(* PLC project RedHat_Demo_MarketingStand_Working.project, CODESYS CODESYS V3.5 SP22 *)
(* stored: creationDateTime 2026-08-06T19:18:19.3184089, modificationDateTime 2026-08-06T19:18:02.9898727 *)

PROGRAM PLC_PRG
  VAR
    Cmd_Run : BOOL;
    R_TRIG_0 : R_TRIG;
    Sequence_Run : DINT := 0;
    Sts_SequenceDone : BOOL;
    Sts_FirstScanBit : BOOL := TRUE;
    TON_MotorDataDelay : ARRAY[0..9] OF TON;
    TON_IndexPauseDelay : TON;
    Par_IndexPause : TIME := TIME#1s0ms;
    TON_Timeout_Reset : TON;
    TON_Timeout_Enable : TON;
    TON_Timeout_Move1 : TON;
    TON_Timeout_Move2 : TON;
    TON_Timeout_Stop : TON;
    Sts_SeqTimeout : DINT;
    Force_Run : BOOL;
    Force_Stop : BOOL;
    Cmd_Stop : BOOL;
    Par_SingleIndex : BOOL;
    TimeStart1 : LTIME;
    tDelta : TIME;
    tStart : TIME;
    tEnd : TIME;
    Return_Time_Input : BOOL;
    ReturnTimeFinish : BOOL;
    MoveDelta : BOOL;
    newTimeDelta : TIME;
    IndexPauseInt : REAL;
    IndexPauseMin : REAL := 500;
    IndexPauseMax : REAL := 5000;
    RealTimeDelta : REAL;
    microtime : SYSTIME;
    Seq0 : BOOL;
    Seq10 : BOOL;
    Seq20 : BOOL;
    Seq30 : BOOL;
    Seq40 : BOOL;
    Seq50 : BOOL;
    Seq60 : BOOL;
    SeqErr : BOOL;
    MotorEnabled : BOOL;
    SeqStop : BOOL;
    SeqMov1 : BOOL;
    SeqMov2 : BOOL;
  END_VAR
  VAR  (* added by the conversion: wires and edge detectors of the diagram *)
    _NE7_OUT : BOOL;
    _EQ14_ENO : BOOL;
    _EQ14_OUT : BOOL;
    _w20 : BOOL;
    _w21 : BOOL;
    _EQ27_ENO : BOOL;
    _EQ27_OUT : BOOL;
    _EQ35_OUT : BOOL;
    _EQ48_OUT : BOOL;
    _EQ65_OUT : BOOL;
    _EQ76_OUT : BOOL;
    _EQ93_OUT : BOOL;
    _EQ113_OUT : BOOL;
    _EQ130_OUT : BOOL;
    _MOVE138_EN : BOOL;
    _EQ145_OUT : BOOL;
    _MOVE162_EN : BOOL;
    R_TRIG1 : R_TRIG;
    R_TRIG2 : R_TRIG;
    _FUNC_SCALE196_EN : BOOL;
  END_VAR

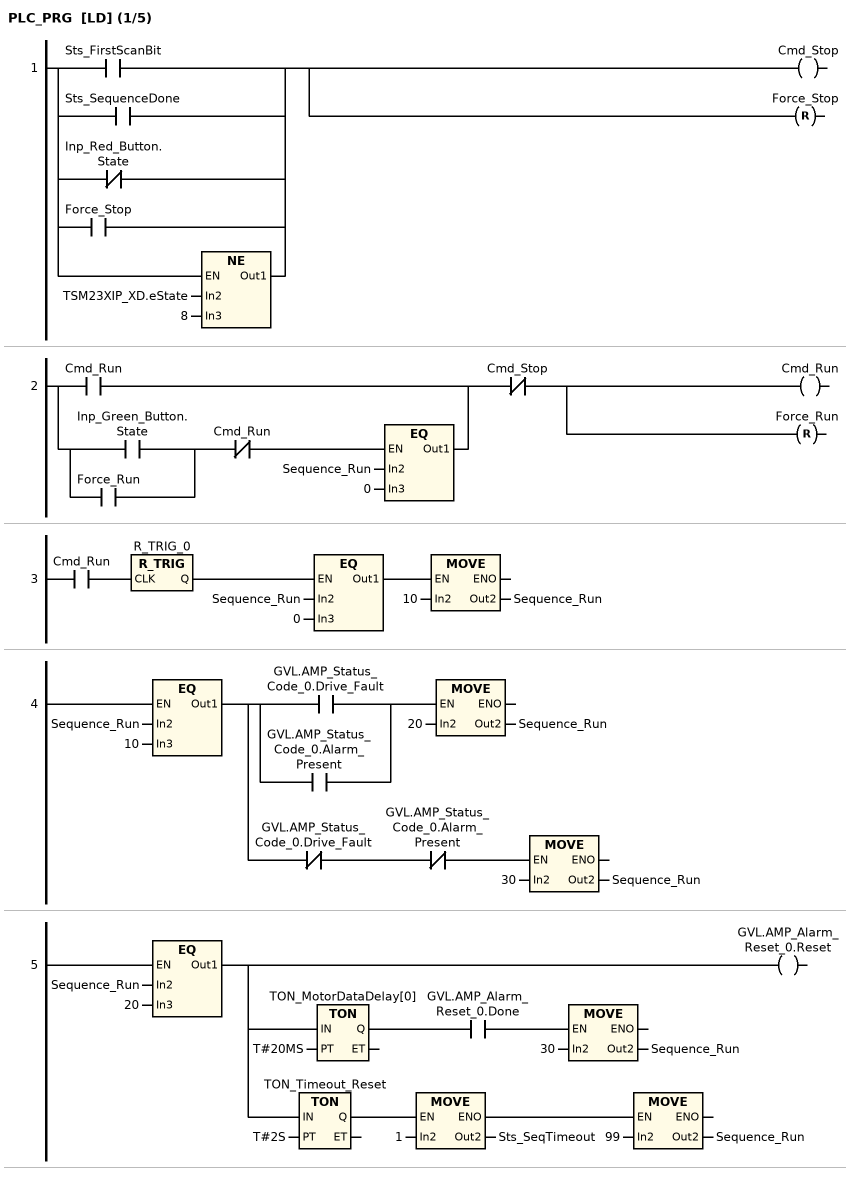
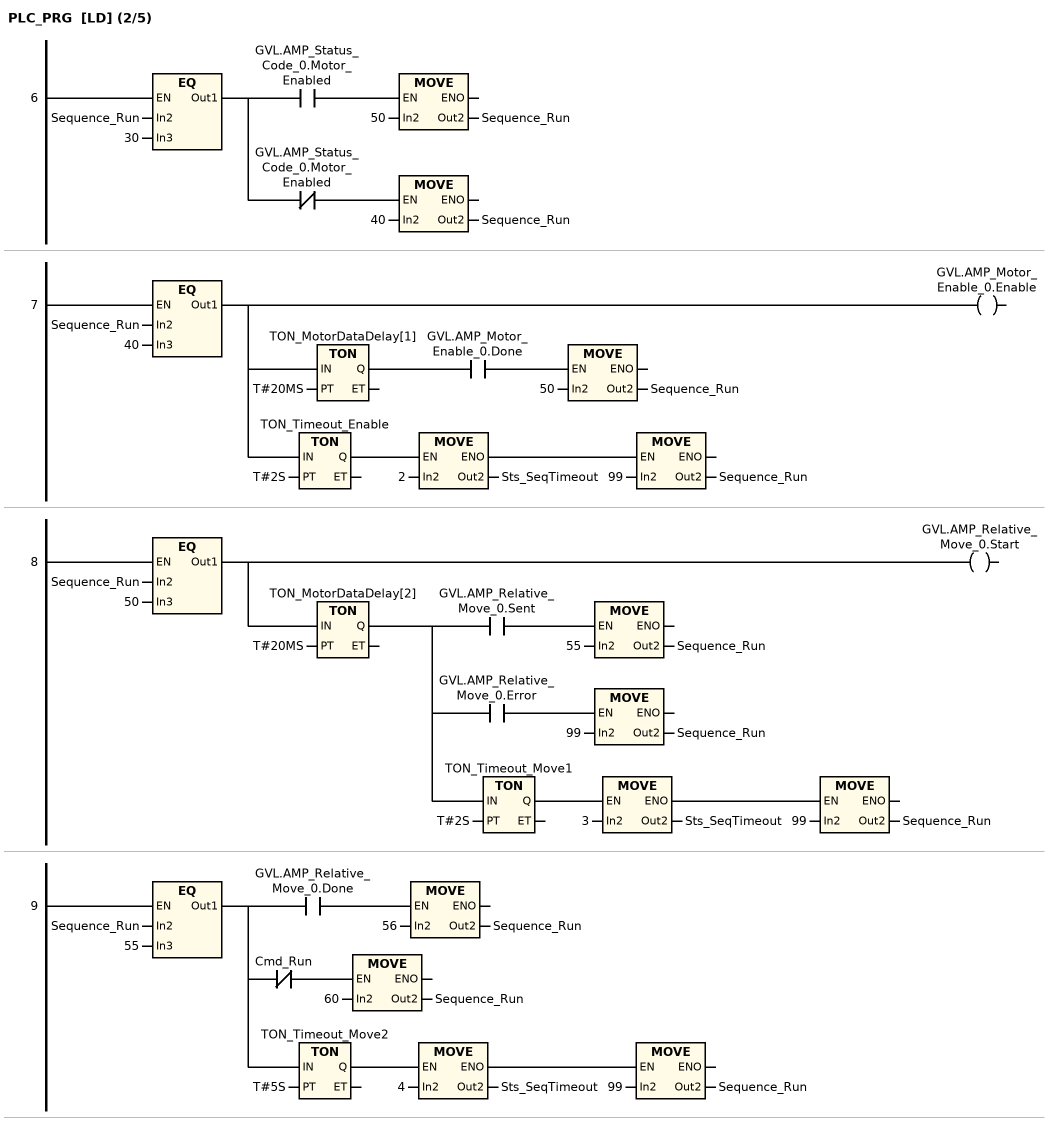
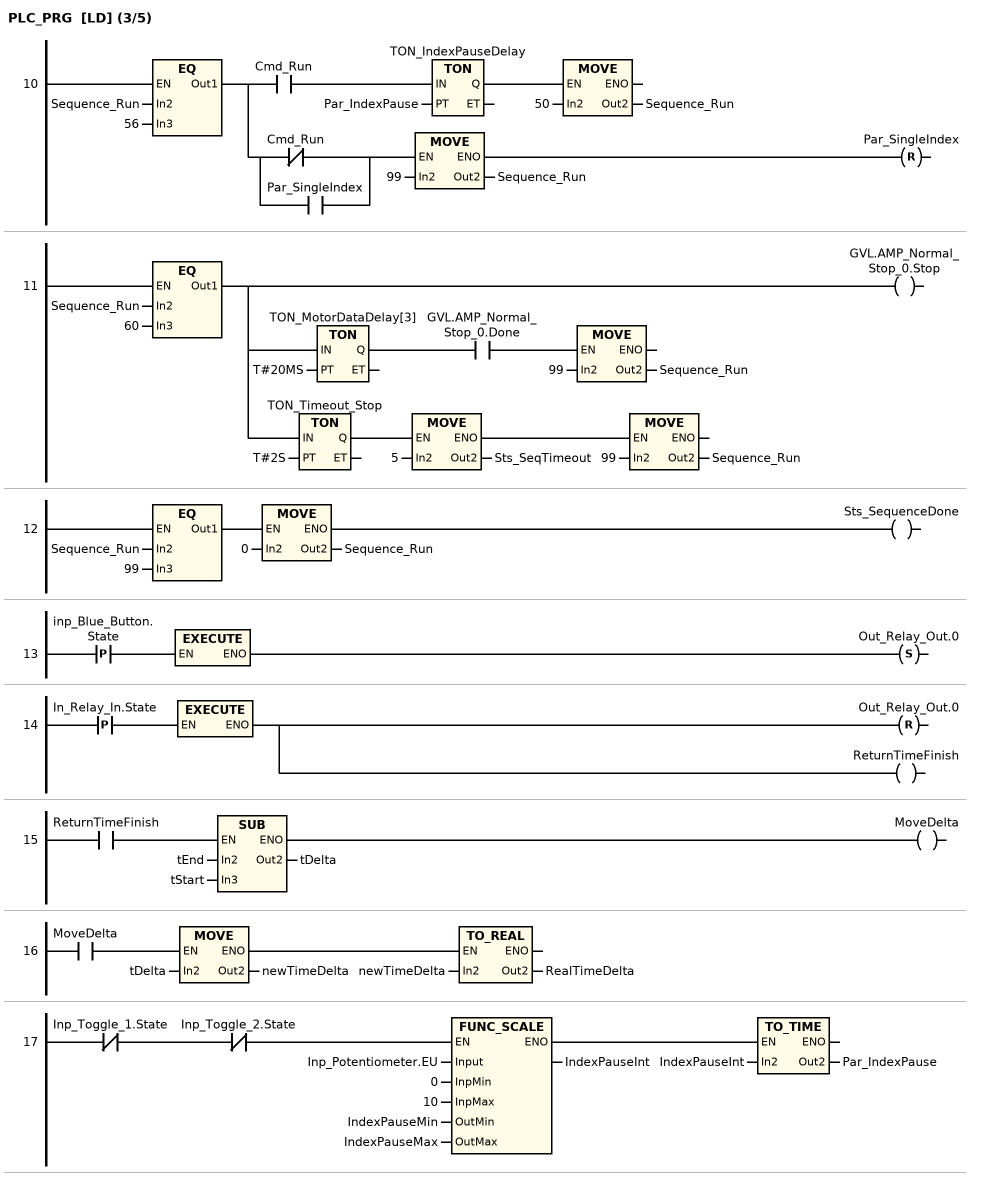
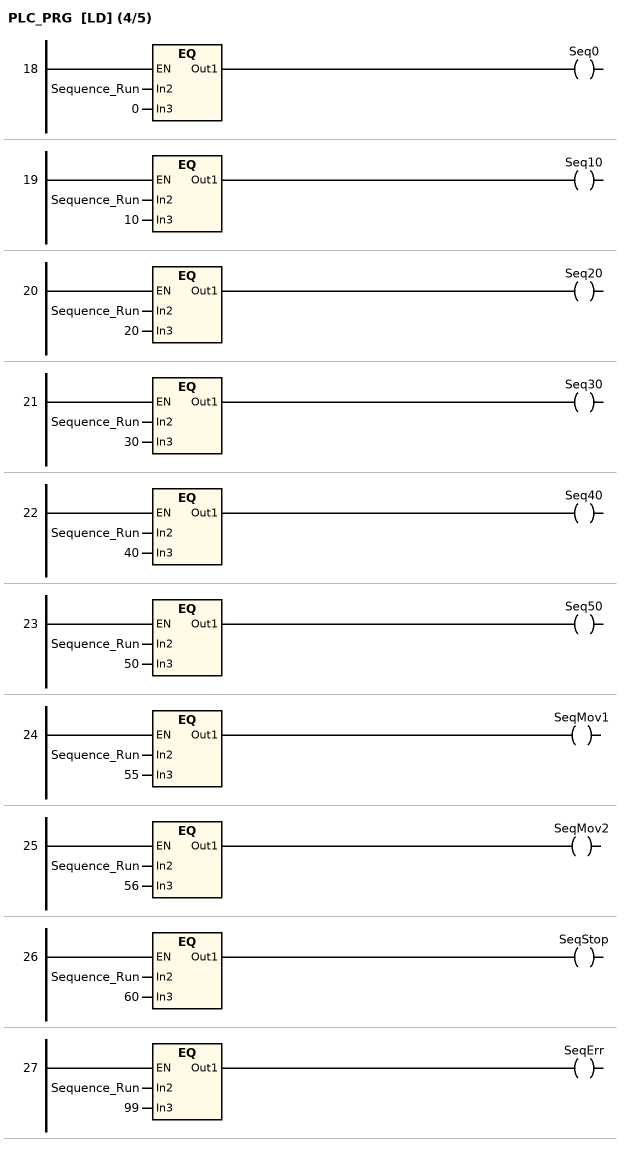
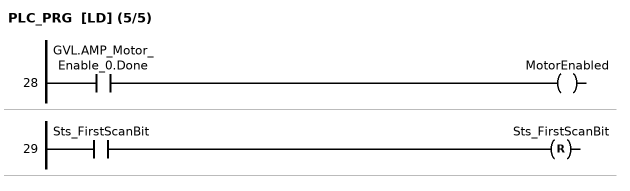
(* LD diagram, written out as Structured Text *)
(* Run Permissives *)

_NE7_OUT := TSM23XIP_XD.eState <> 8;
Cmd_Stop := Sts_FirstScanBit OR Sts_SequenceDone OR NOT Inp_Red_Button.State OR Force_Stop OR _NE7_OUT;
IF Sts_FirstScanBit OR Sts_SequenceDone OR NOT Inp_Red_Button.State OR Force_Stop OR _NE7_OUT THEN Force_Stop := FALSE; END_IF;
(* Start Sequence Command *)

_EQ14_OUT := EQ(EN := (Inp_Green_Button.State OR Force_Run) AND NOT Cmd_Run, IN1 := Sequence_Run, IN2 := 0, ENO => _EQ14_ENO);
_w20 := Cmd_Run;
_w21 := (_EQ14_OUT OR _w20) AND NOT Cmd_Stop;
Cmd_Run := _w21;
IF _w21 THEN Force_Run := FALSE; END_IF;

R_TRIG_0(CLK := Cmd_Run);
_EQ27_OUT := EQ(EN := R_TRIG_0.Q, IN1 := Sequence_Run, IN2 := 0, ENO => _EQ27_ENO);
IF _EQ27_OUT THEN Sequence_Run := 10; END_IF;

_EQ35_OUT := Sequence_Run = 10;
IF _EQ35_OUT AND NOT GVL.AMP_Status_Code_0.Drive_Fault AND NOT GVL.AMP_Status_Code_0.Alarm_Present THEN Sequence_Run := 30; END_IF;
IF _EQ35_OUT AND (GVL.AMP_Status_Code_0.Drive_Fault OR GVL.AMP_Status_Code_0.Alarm_Present) THEN Sequence_Run := 20; END_IF;
(* Fault Reset *)

_EQ48_OUT := Sequence_Run = 20;
GVL.AMP_Alarm_Reset_0.Reset := _EQ48_OUT;
TON_MotorDataDelay[0](IN := _EQ48_OUT, PT := T#20MS);
IF TON_MotorDataDelay[0].Q AND GVL.AMP_Alarm_Reset_0.Done THEN Sequence_Run := 30; END_IF;
TON_Timeout_Reset(IN := _EQ48_OUT, PT := T#2S);
IF TON_Timeout_Reset.Q THEN Sts_SeqTimeout := 1; END_IF;
IF TON_Timeout_Reset.Q THEN Sequence_Run := 99; END_IF;

_EQ65_OUT := Sequence_Run = 30;
IF _EQ65_OUT AND GVL.AMP_Status_Code_0.Motor_Enabled THEN Sequence_Run := 50; END_IF;
IF _EQ65_OUT AND NOT GVL.AMP_Status_Code_0.Motor_Enabled THEN Sequence_Run := 40; END_IF;
(* Energize *)

_EQ76_OUT := Sequence_Run = 40;
GVL.AMP_Motor_Enable_0.Enable := _EQ76_OUT;
TON_MotorDataDelay[1](IN := _EQ76_OUT, PT := T#20MS);
IF TON_MotorDataDelay[1].Q AND GVL.AMP_Motor_Enable_0.Done THEN Sequence_Run := 50; END_IF;
TON_Timeout_Enable(IN := _EQ76_OUT, PT := T#2S);
IF TON_Timeout_Enable.Q THEN Sts_SeqTimeout := 2; END_IF;
IF TON_Timeout_Enable.Q THEN Sequence_Run := 99; END_IF;
(* Incremental Move *)

_EQ93_OUT := Sequence_Run = 50;
GVL.AMP_Relative_Move_0.Start := _EQ93_OUT;
TON_MotorDataDelay[2](IN := _EQ93_OUT, PT := T#20MS);
IF TON_MotorDataDelay[2].Q AND GVL.AMP_Relative_Move_0.Sent THEN Sequence_Run := 55; END_IF;
IF TON_MotorDataDelay[2].Q AND GVL.AMP_Relative_Move_0.Error THEN Sequence_Run := 99; END_IF;
TON_Timeout_Move1(IN := TON_MotorDataDelay[2].Q, PT := T#2S);
IF TON_Timeout_Move1.Q THEN Sts_SeqTimeout := 3; END_IF;
IF TON_Timeout_Move1.Q THEN Sequence_Run := 99; END_IF;
(* Wait For Move To Complete, or Stop button Press *)

_EQ113_OUT := Sequence_Run = 55;
IF _EQ113_OUT AND GVL.AMP_Relative_Move_0.Done THEN Sequence_Run := 56; END_IF;
IF _EQ113_OUT AND NOT Cmd_Run THEN Sequence_Run := 60; END_IF;
TON_Timeout_Move2(IN := _EQ113_OUT, PT := T#5S);
IF TON_Timeout_Move2.Q THEN Sts_SeqTimeout := 4; END_IF;
IF TON_Timeout_Move2.Q THEN Sequence_Run := 99; END_IF;
(* Pause before next index (Loop Up) *)

_EQ130_OUT := Sequence_Run = 56;
TON_IndexPauseDelay(IN := _EQ130_OUT AND Cmd_Run, PT := Par_IndexPause);
IF TON_IndexPauseDelay.Q THEN Sequence_Run := 50; END_IF;
_MOVE138_EN := _EQ130_OUT AND (NOT Cmd_Run OR Par_SingleIndex);
IF _MOVE138_EN THEN Sequence_Run := 99; END_IF;
IF _MOVE138_EN THEN Par_SingleIndex := FALSE; END_IF;
(* Normal Stop *)

_EQ145_OUT := Sequence_Run = 60;
GVL.AMP_Normal_Stop_0.Stop := _EQ145_OUT;
TON_MotorDataDelay[3](IN := _EQ145_OUT, PT := T#20MS);
IF TON_MotorDataDelay[3].Q AND GVL.AMP_Normal_Stop_0.Done THEN Sequence_Run := 99; END_IF;
TON_Timeout_Stop(IN := _EQ145_OUT, PT := T#2S);
IF TON_Timeout_Stop.Q THEN Sts_SeqTimeout := 5; END_IF;
IF TON_Timeout_Stop.Q THEN Sequence_Run := 99; END_IF;
(* Sequence Complete *)

_MOVE162_EN := Sequence_Run = 99;
IF _MOVE162_EN THEN Sequence_Run := 0; END_IF;
Sts_SequenceDone := _MOVE162_EN;

R_TRIG1(CLK := inp_Blue_Button.State);
IF R_TRIG1.Q THEN
  tStart := TO_TIME(SysTimeGetMs());
END_IF;
IF R_TRIG1.Q THEN Out_Relay_Out.0 := TRUE; END_IF;

R_TRIG2(CLK := In_Relay_In.State);
IF R_TRIG2.Q THEN
  tEnd := TO_TIME(SysTimeGetMs());
END_IF;
IF R_TRIG2.Q THEN Out_Relay_Out.0 := FALSE; END_IF;
ReturnTimeFinish := R_TRIG2.Q;

IF ReturnTimeFinish THEN tDelta := tEnd - tStart; END_IF;
MoveDelta := ReturnTimeFinish;

IF MoveDelta THEN newTimeDelta := tDelta; END_IF;
IF MoveDelta THEN RealTimeDelta := TO_REAL(In2 := newTimeDelta); END_IF;

_FUNC_SCALE196_EN := NOT Inp_Toggle_1.State AND NOT Inp_Toggle_2.State;
IF _FUNC_SCALE196_EN THEN IndexPauseInt := FUNC_SCALE(Input := Inp_Potentiometer.EU, InpMin := 0, InpMax := 10, OutMin := IndexPauseMin, OutMax := IndexPauseMax); END_IF;
IF _FUNC_SCALE196_EN THEN Par_IndexPause := TO_TIME(In2 := IndexPauseInt); END_IF;

Seq0 := Sequence_Run = 0;

Seq10 := Sequence_Run = 10;

Seq20 := Sequence_Run = 20;

Seq30 := Sequence_Run = 30;

Seq40 := Sequence_Run = 40;

Seq50 := Sequence_Run = 50;

SeqMov1 := Sequence_Run = 55;

SeqMov2 := Sequence_Run = 56;


SeqStop := Sequence_Run = 60;

SeqErr := Sequence_Run = 99;

MotorEnabled := GVL.AMP_Motor_Enable_0.Done;

(* Turn off First Scan Bit *)

IF Sts_FirstScanBit THEN Sts_FirstScanBit := FALSE; END_IF;
END_PROGRAM

FUNCTION FUNC_SCALE : REAL
  VAR_INPUT
    Input : REAL;
    InpMin : REAL;
    InpMax : REAL;
    OutMin : REAL;
    OutMax : REAL;
  END_VAR
  VAR
    Value : REAL;
  END_VAR

                    IF Input < InpMin THEN
	Value:= InpMin;
ELSIF Input > InpMax THEN
	Value:= InpMax;
ELSE
	Value:= Input;
END_IF
FUNC_SCALE:= (Value-InpMin) * (OutMax-OutMin) / (InpMax-InpMin) + OutMin;
                  
END_FUNCTION

PROGRAM MOTOR
  VAR CONSTANT
    StepsPerRotation : REAL := 20000;
  END_VAR
  VAR
    Par_SelectorDistance1_Degrees : REAL := -30;  (* Motor Distance variables corresponding to the 3 positions of the selector switch, in degrees. Code converts to steps *)
    Par_SelectorDistance2_Degrees : REAL := 30;
    Par_SelectorDistance3_Degrees : REAL := 60;
    Par_SoftwareDistanceEnable : BOOL;  (* If want to ignore selector switch and use software Distance value *)
    Par_SoftwareDistance_Degrees : REAL;
    MotorDistance_Steps : REAL;  (* Calculated steps to send to motor *)
    Par_PotentiometerMinSpeed : REAL := 0.2;  (* Potentiometer used for index speed. Set minimum and maximum *)
    Par_PotentiometerMaxSpeed : REAL := 0.3;
    Par_AccelDeccel : REAL := 0.167;  (* Constant acceleration and deceleration *)
    Par_SoftwareSpeedEnable : BOOL;  (* If want to ignore potentiometer and use software Speed value *)
    Par_SoftwareSpeed : REAL;
    EncoderPosition_Degrees : REAL;  (* Calculated Position In Degrees of the encoder *)
    Par_SCL_Reg1 : DINT;
    Cmd_ZeroPosition : BOOL;  (* Zero Position Sequence *)
    Sequence_ZeroPosition : DINT;
    TON_MotorDataDelay : ARRAY[0..1] OF TON;
  END_VAR
  VAR  (* added by the conversion: wires and edge detectors of the diagram *)
    _GT46_ENO : BOOL;
    _GT46_OUT : BOOL;
    _EQ103_ENO : BOOL;
    _EQ103_OUT : BOOL;
    _EQ111_OUT : BOOL;
    _EQ121_OUT : BOOL;
    _EQ129_OUT : BOOL;
    _EQ139_OUT : BOOL;
  END_VAR

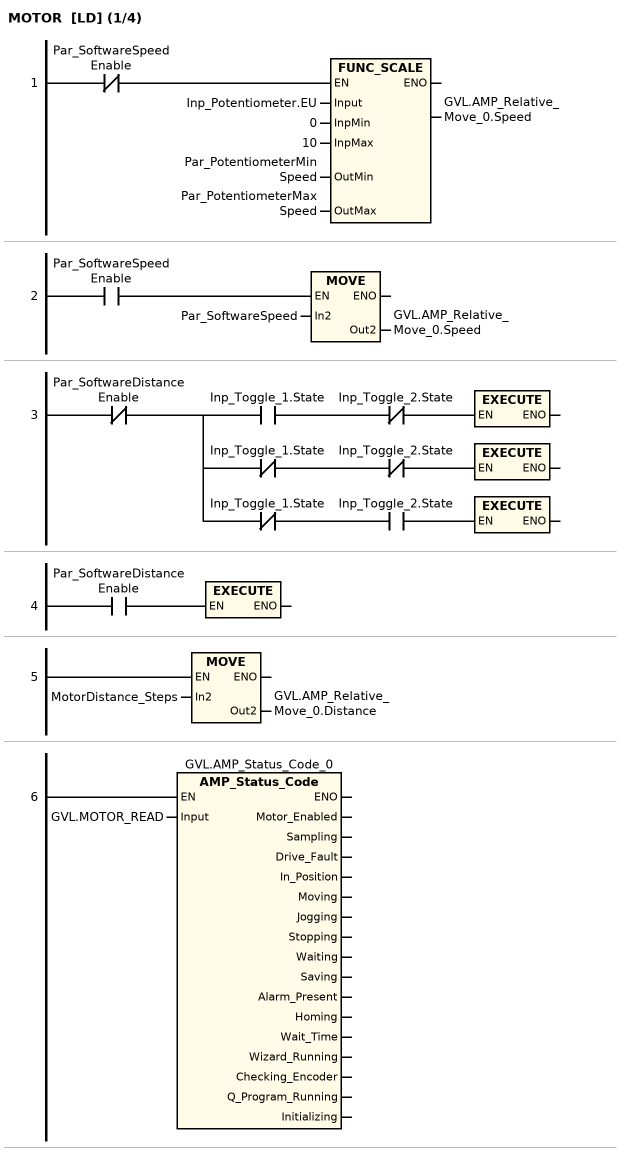
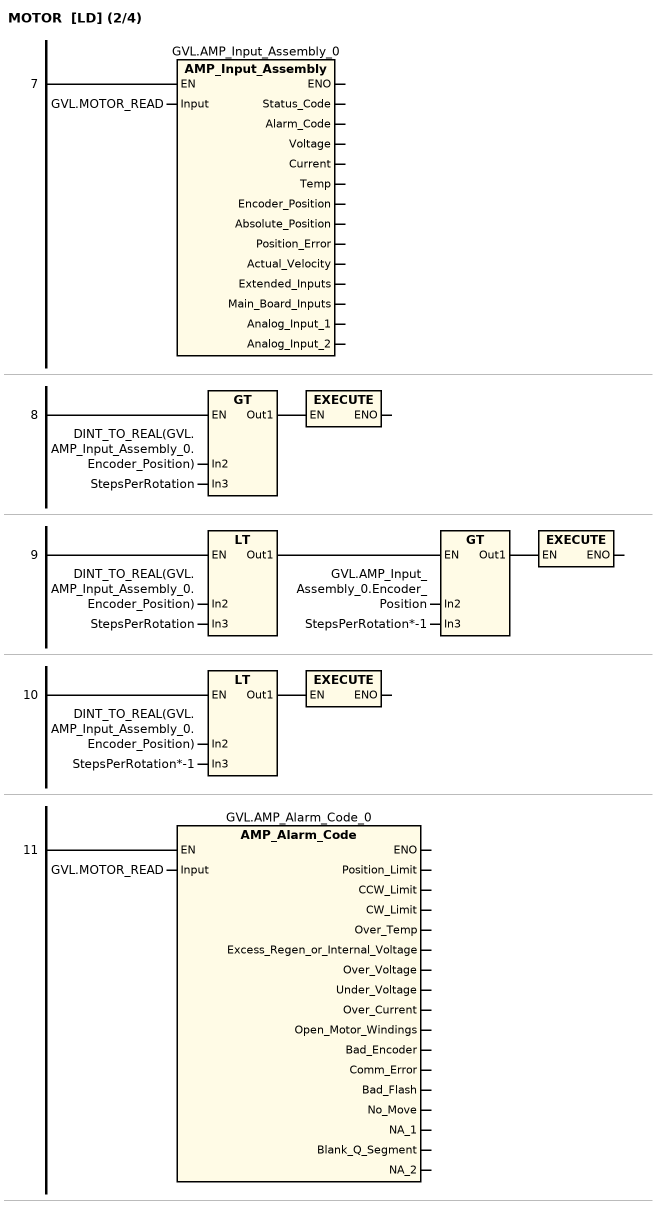
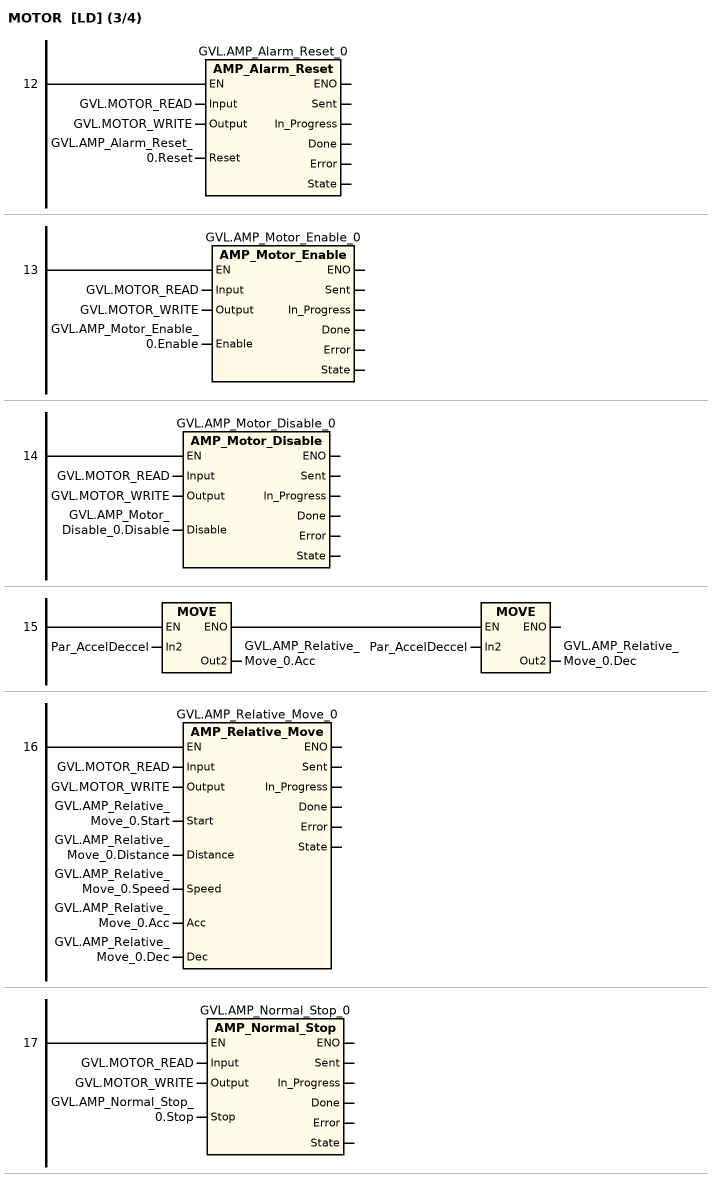
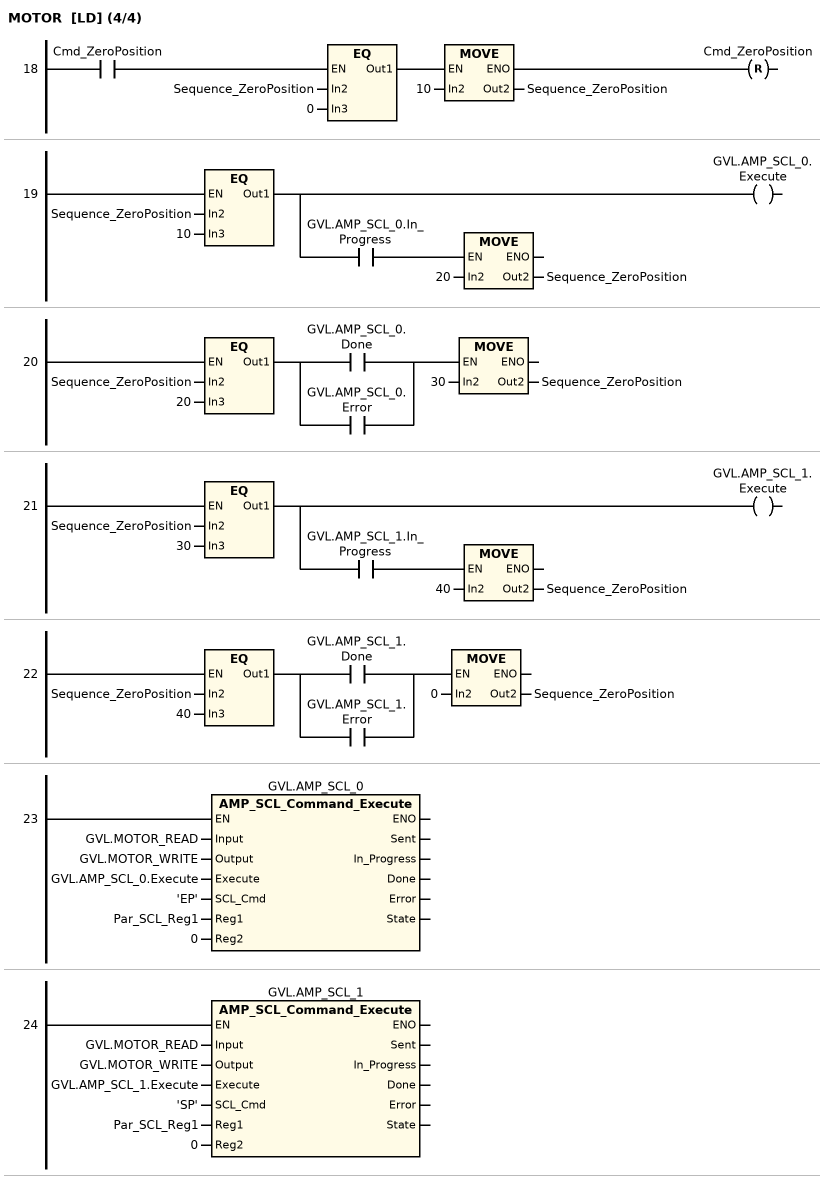
(* LD diagram, written out as Structured Text *)
(* Scale Move speed from Potentiometer *)

IF NOT Par_SoftwareSpeedEnable THEN GVL.AMP_Relative_Move_0.Speed := FUNC_SCALE(Input := Inp_Potentiometer.EU, InpMin := 0, InpMax := 10, OutMin := Par_PotentiometerMinSpeed, OutMax := Par_PotentiometerMaxSpeed); END_IF;
IF Par_SoftwareSpeedEnable THEN GVL.AMP_Relative_Move_0.Speed := Par_SoftwareSpeed; END_IF;

(* Set Move Distance from Toggle Switch. Convert Degrees to steps *)

IF NOT Par_SoftwareDistanceEnable AND Inp_Toggle_1.State AND NOT Inp_Toggle_2.State THEN
  MotorDistance_Steps:= Par_SelectorDistance1_Degrees / 360 * StepsPerRotation;
END_IF;
IF NOT Par_SoftwareDistanceEnable AND NOT Inp_Toggle_1.State AND NOT Inp_Toggle_2.State THEN
  MotorDistance_Steps:= Par_SelectorDistance2_Degrees / 360 * StepsPerRotation;
END_IF;
IF NOT Par_SoftwareDistanceEnable AND NOT Inp_Toggle_1.State AND Inp_Toggle_2.State THEN
  MotorDistance_Steps:= Par_SelectorDistance3_Degrees / 360 * StepsPerRotation;
END_IF;
IF Par_SoftwareDistanceEnable THEN
  MotorDistance_Steps:= Par_SoftwareDistance_Degrees / 360 * StepsPerRotation;
END_IF;
GVL.AMP_Relative_Move_0.Distance := MotorDistance_Steps;
(* Motor Functions *)

GVL.AMP_Status_Code_0(Input := GVL.MOTOR_READ);

GVL.AMP_Input_Assembly_0(Input := GVL.MOTOR_READ);
(* Calculate Position Degrees based on Encoder Position. *)

IF DINT_TO_REAL(GVL.AMP_Input_Assembly_0.Encoder_Position) > StepsPerRotation THEN
  EncoderPosition_Degrees:= OSCAT_BASIC.MODR(IN:= DINT_TO_REAL(GVL.AMP_Input_Assembly_0.Encoder_Position), DIVI:= StepsPerRotation)/20000*360;
END_IF;
_GT46_OUT := GT(EN := DINT_TO_REAL(GVL.AMP_Input_Assembly_0.Encoder_Position) < StepsPerRotation, IN1 := GVL.AMP_Input_Assembly_0.Encoder_Position, IN2 := StepsPerRotation*-1, ENO => _GT46_ENO);
IF _GT46_OUT THEN
  EncoderPosition_Degrees:= DINT_TO_REAL(GVL.AMP_Input_Assembly_0.Encoder_Position) / StepsPerRotation * 360;
END_IF;
IF DINT_TO_REAL(GVL.AMP_Input_Assembly_0.Encoder_Position) < (StepsPerRotation*-1) THEN
  EncoderPosition_Degrees:= ABS(OSCAT_BASIC.MODR(IN:= DINT_TO_REAL(GVL.AMP_Input_Assembly_0.Encoder_Position), DIVI:= StepsPerRotation))/20000*360;
END_IF;

GVL.AMP_Alarm_Code_0(Input := GVL.MOTOR_READ);

GVL.AMP_Alarm_Reset_0(Input := GVL.MOTOR_READ, Output := GVL.MOTOR_WRITE, Reset := GVL.AMP_Alarm_Reset_0.Reset);

GVL.AMP_Motor_Enable_0(Input := GVL.MOTOR_READ, Output := GVL.MOTOR_WRITE, Enable := GVL.AMP_Motor_Enable_0.Enable);

GVL.AMP_Motor_Disable_0(Input := GVL.MOTOR_READ, Output := GVL.MOTOR_WRITE, Disable := GVL.AMP_Motor_Disable_0.Disable);

GVL.AMP_Relative_Move_0.Acc := Par_AccelDeccel;
GVL.AMP_Relative_Move_0.Dec := Par_AccelDeccel;

GVL.AMP_Relative_Move_0(Input := GVL.MOTOR_READ, Output := GVL.MOTOR_WRITE, Start := GVL.AMP_Relative_Move_0.Start, Distance := GVL.AMP_Relative_Move_0.Distance, Speed := GVL.AMP_Relative_Move_0.Speed, Acc := GVL.AMP_Relative_Move_0.Acc, Dec := GVL.AMP_Relative_Move_0.Dec);

GVL.AMP_Normal_Stop_0(Input := GVL.MOTOR_READ, Output := GVL.MOTOR_WRITE, Stop := GVL.AMP_Normal_Stop_0.Stop);
(* Sequence to Zero the encoder position. Requires manual toggle. *)

_EQ103_OUT := EQ(EN := Cmd_ZeroPosition, IN1 := Sequence_ZeroPosition, IN2 := 0, ENO => _EQ103_ENO);
IF _EQ103_OUT THEN Sequence_ZeroPosition := 10; END_IF;
IF _EQ103_OUT THEN Cmd_ZeroPosition := FALSE; END_IF;

_EQ111_OUT := Sequence_ZeroPosition = 10;
GVL.AMP_SCL_0.Execute := _EQ111_OUT;
IF _EQ111_OUT AND GVL.AMP_SCL_0.In_Progress THEN Sequence_ZeroPosition := 20; END_IF;

_EQ121_OUT := Sequence_ZeroPosition = 20;
IF _EQ121_OUT AND (GVL.AMP_SCL_0.Done OR GVL.AMP_SCL_0.Error) THEN Sequence_ZeroPosition := 30; END_IF;

_EQ129_OUT := Sequence_ZeroPosition = 30;
GVL.AMP_SCL_1.Execute := _EQ129_OUT;
IF _EQ129_OUT AND GVL.AMP_SCL_1.In_Progress THEN Sequence_ZeroPosition := 40; END_IF;

_EQ139_OUT := Sequence_ZeroPosition = 40;
IF _EQ139_OUT AND (GVL.AMP_SCL_1.Done OR GVL.AMP_SCL_1.Error) THEN Sequence_ZeroPosition := 0; END_IF;

GVL.AMP_SCL_0(Input := GVL.MOTOR_READ, Output := GVL.MOTOR_WRITE, Execute := GVL.AMP_SCL_0.Execute, SCL_Cmd := 'EP', Reg1 := Par_SCL_Reg1, Reg2 := 0);

GVL.AMP_SCL_1(Input := GVL.MOTOR_READ, Output := GVL.MOTOR_WRITE, Execute := GVL.AMP_SCL_1.Execute, SCL_Cmd := 'SP', Reg1 := Par_SCL_Reg1, Reg2 := 0);
END_PROGRAM

PROGRAM LIGHT_CYCLE
  VAR
    TON_0 : TON;
    Cmd_Light : INT;
    RedStack : BOOL;
    YellowStack : BOOL;
    GreenStack : BOOL;
    BlueButton : BOOL;
    RedButton : BOOL;
    GreenButton : BOOL;
  END_VAR
  VAR  (* added by the conversion: wires and edge detectors of the diagram *)
    _EQ4_ENO : BOOL;
    _EQ4_OUT : BOOL;
    _EQ16_OUT : BOOL;
    _EQ23_OUT : BOOL;
    _EQ30_OUT : BOOL;
  END_VAR

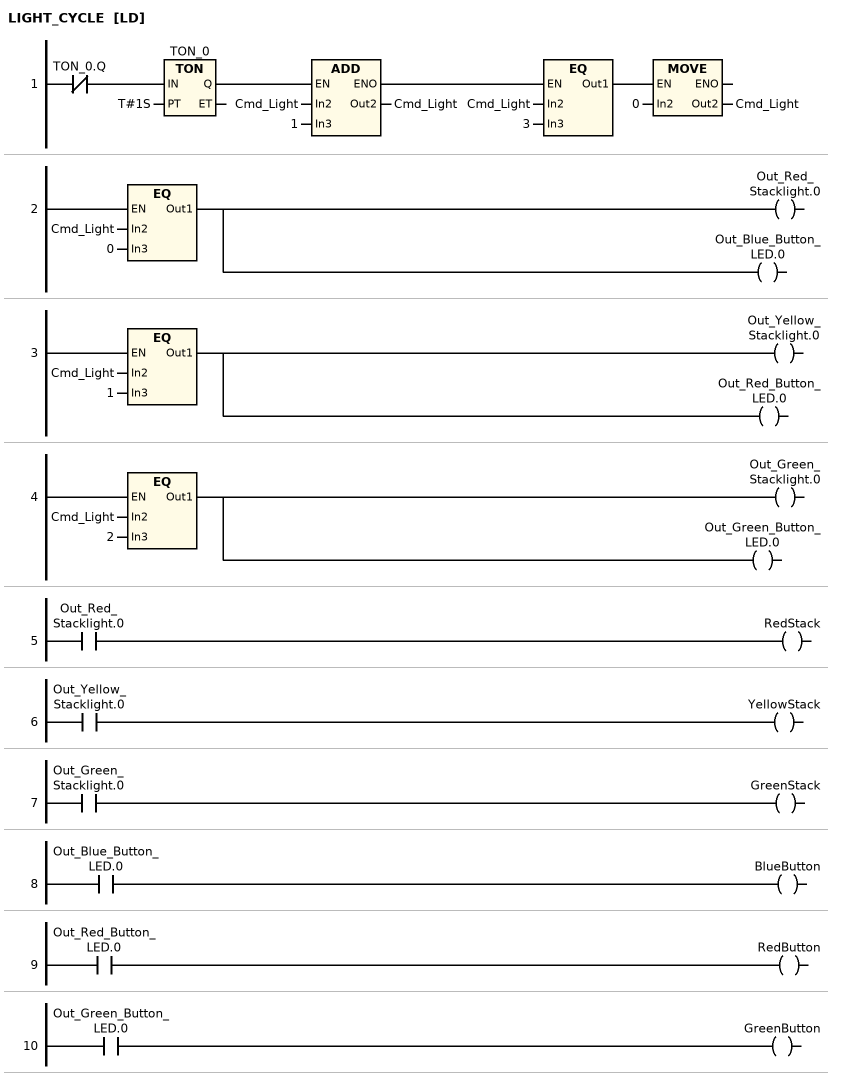
(* LD diagram, written out as Structured Text *)

TON_0(IN := NOT TON_0.Q, PT := T#1S);
IF TON_0.Q THEN Cmd_Light := Cmd_Light + 1; END_IF;
_EQ4_OUT := EQ(EN := TON_0.Q, IN1 := Cmd_Light, IN2 := 3, ENO => _EQ4_ENO);
IF _EQ4_OUT THEN Cmd_Light := 0; END_IF;

_EQ16_OUT := Cmd_Light = 0;
Out_Red_Stacklight.0 := _EQ16_OUT;
Out_Blue_Button_LED.0 := _EQ16_OUT;

_EQ23_OUT := Cmd_Light = 1;
Out_Yellow_Stacklight.0 := _EQ23_OUT;
Out_Red_Button_LED.0 := _EQ23_OUT;

_EQ30_OUT := Cmd_Light = 2;
Out_Green_Stacklight.0 := _EQ30_OUT;
Out_Green_Button_LED.0 := _EQ30_OUT;

RedStack := Out_Red_Stacklight.0;

YellowStack := Out_Yellow_Stacklight.0;

GreenStack := Out_Green_Stacklight.0;

BlueButton := Out_Blue_Button_LED.0;

RedButton := Out_Red_Button_LED.0;

GreenButton := Out_Green_Button_LED.0;
END_PROGRAM

CONFIGURATION Device
  RESOURCE Application ON PLC
    {attribute 'qualified_only'}
    VAR_GLOBAL  (* GVL *)
      MOTOR_READ : ARRAY[0..13] OF DINT;  (* Motor Function Variables *)
      MOTOR_WRITE : ARRAY[0..15] OF DINT;
      AMP_Status_Code_0 : AMP_Status_Code;
      AMP_Input_Assembly_0 : AMP_Input_Assembly;
      AMP_Alarm_Code_0 : AMP_Alarm_Code;
      AMP_Alarm_Reset_0 : AMP_Alarm_Reset;
      AMP_Motor_Enable_0 : AMP_Motor_Enable;
      AMP_Motor_Disable_0 : AMP_Motor_Disable;
      AMP_Relative_Move_0 : AMP_Relative_Move;
      AMP_Normal_Stop_0 : AMP_Normal_Stop;
      AMP_SCL_0 : AMP_SCL_Command_Execute;
      AMP_SCL_1 : AMP_SCL_Command_Execute;
    END_VAR
    TASK MainTask(INTERVAL := T#10ms, PRIORITY := 2);
    TASK ENIPScannerIOTask(INTERVAL := T#10ms, PRIORITY := 0);
    TASK ENIPScannerServiceTask(INTERVAL := T#20ms, PRIORITY := 30);
    PROGRAM MOTOR WITH MainTask : MOTOR;
    PROGRAM PLC_PRG WITH MainTask : PLC_PRG;
    PROGRAM LIGHT_CYCLE WITH MainTask : LIGHT_CYCLE;
    PROGRAM EtherNet_IP_Scanner.IOCycle WITH ENIPScannerIOTask : EtherNet_IP_Scanner.IOCycle;
    PROGRAM EtherNet_IP_Scanner.ServiceCycle WITH ENIPScannerServiceTask : EtherNet_IP_Scanner.ServiceCycle;
  END_RESOURCE
END_CONFIGURATION

CONFIGURATION Ethernet
END_CONFIGURATION

CONFIGURATION EtherNet_IP_Scanner
END_CONFIGURATION

CONFIGURATION TSM23XIP_XD
END_CONFIGURATION

CONFIGURATION Opto22_RIO1
END_CONFIGURATION

CONFIGURATION Red_Button_LED
END_CONFIGURATION

CONFIGURATION Green_Button_LED
END_CONFIGURATION

CONFIGURATION Blue_Button_LED
END_CONFIGURATION

CONFIGURATION Red_Button
END_CONFIGURATION

CONFIGURATION Green_Button
END_CONFIGURATION

CONFIGURATION Blue_Button
END_CONFIGURATION

CONFIGURATION Relay_In
END_CONFIGURATION

CONFIGURATION <Empty7>
END_CONFIGURATION

CONFIGURATION Relay_Out
END_CONFIGURATION

CONFIGURATION <Empty9>
END_CONFIGURATION

CONFIGURATION Opto22_RIO2
END_CONFIGURATION

CONFIGURATION Red_Stacklight
END_CONFIGURATION

CONFIGURATION Yellow_Stacklight
END_CONFIGURATION

CONFIGURATION Green_Stacklight
END_CONFIGURATION

CONFIGURATION Toggle_1
END_CONFIGURATION

CONFIGURATION Toggle_2
END_CONFIGURATION

CONFIGURATION Potentiometer
END_CONFIGURATION

CONFIGURATION <Empty6>
END_CONFIGURATION

CONFIGURATION <Empty7>
END_CONFIGURATION

CONFIGURATION <Empty8>
END_CONFIGURATION

CONFIGURATION <Empty9>
END_CONFIGURATION
